PROGRAM prgComEffIO
VAR
	fbCom			: FB_MqttCommunicator_V2;
END_VAR

fbCom(
	bConnect:= TRUE,
	strAuthKey :='EIO08031879806',
	sUserName:= '90b3d39e-7421-4c3d-851d-5bcf1221f0e6', 
	sUserPassword:= 'f8bcb488-dc42-4c36-ba45-df0dd9149713', 
	eSavePositionCertificate:= eSavePositionOnPLC.ePostionHardDisk,
	time_HeartBeat_sec	:= T#15S, 
	bConnected=> , 
	bError=> , 
	hrErrorCode=> , 
	eConnectionState=> , 
	eErrorMessage_Out=> );

END_PROGRAM

(* stored: Version 1.1.0.1, ProductVersion 3.1.4024.11
   POU prgComEffIO: Id {e6a8073a-1427-4947-b617-9ed5a73dda57}, SpecialFunc None *)
